TYPE DoDiag :
STRUCT
	{attribute addProperty Name "Diag"}
	Diag AT %I* : BOOL;
END_STRUCT
END_TYPE

(* stored: Version 1.1.0.1, ProductVersion 3.1.4024.9
   DUT DoDiag: Id {1448db76-bb3f-084b-07cf-2f4f0bd875c5} *)
